RoboDK station: Project_AutomationPipeCouplingArm_Full.rdk

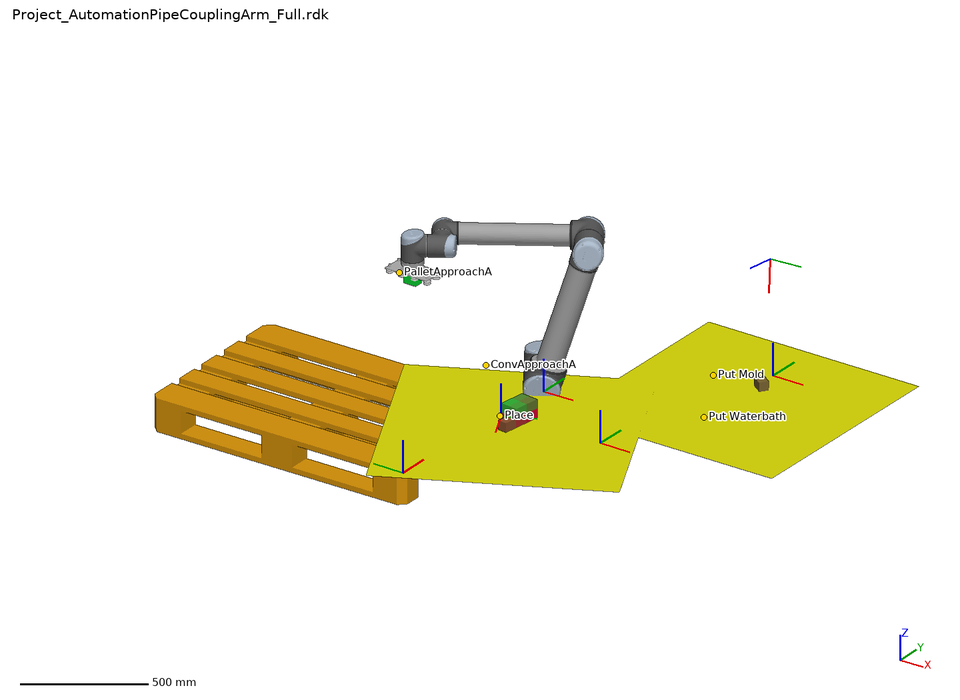
[picture v0: the station drawn from its stored meshes, robots at their saved joint values, targets as dots, program paths as lines]
Station Project_AutomationPipeCouplingArm_Full (saved by RoboDK 5.9.0). Poses are relative to the parent item; angles as X-Y-Z fixed-axis rotations.
Station parameters (name, value as stored): SizeBox, 40, 60, 40, SizePallet, 2,3,2, ConvSpeed, 15.0, SENSOR, 0
  - frame UR10 Base A at (0, -212.57, -10) mm
    - robot UR10 A: 6 axes, payload 10 kg, reach 1300 mm, repeatability 0.1 mm, weight 28.9 kg
        modified DH rows (alpha deg, a mm, theta deg, d mm): 0, 0, 0, 118; 90, 0, 180, 0; 0, 612.7, 0, 0; 0, 571.6, 0, 163.9; -90, 0, 0, 115.7; 90, 0, 180, 92.2
        joint limits [-360, -360, -360, -360, -360, -360] to [360, 360, 360, 360, 360, 360]; home [0, -90, 90, -90, -90, 0]; saved at [33.215, -107.184, 106.915, -89.731, -90, -55.617]
      - tool GripperA, TCP at (0, 0, 30) mm, rotated rx 0 ry 0 rz 90 deg, size 209.9 x 42 x 100 mm, geometry from test.iges
        - object Part 12 at (0, 0, 20) mm, rotated rx -180 ry 0 rz 0 deg, size 40 x 60 x 40 mm, geometry from box.sld
      - tool TCP A, TCP at (0, 0, 50) mm, rotated rx 0 ry 0 rz 90 deg
      - tool TCP A, TCP at (0, 0, 50) mm, rotated rx 0 ry 0 rz 90 deg
      - tool TCP A, TCP at (0, 0, 50) mm, rotated rx 0 ry 0 rz 90 deg
      - tool TCP A, TCP at (0, 0, 50) mm, rotated rx 0 ry 0 rz 90 deg
      - tool TCP A, TCP at (0, 0, 50) mm, rotated rx 0 ry 0 rz 90 deg
      - tool TCP A, TCP at (0, 0, 50) mm, rotated rx 0 ry 0 rz 90 deg
      - tool TCP A, TCP at (0, 0, 50) mm, rotated rx 0 ry 0 rz 90 deg
      - tool TCP A, TCP at (0, 0, 50) mm, rotated rx 0 ry 0 rz 90 deg
      - tool TCP A, TCP at (0, 0, 50) mm, rotated rx 0 ry 0 rz 90 deg
      - tool TCP A, TCP at (0, 0, 50) mm, rotated rx 0 ry 0 rz 90 deg
      - tool TCP A, TCP at (0, 0, 50) mm, rotated rx 0 ry 0 rz 90 deg
      - tool TCP A, TCP at (0, 0, 50) mm, rotated rx 0 ry 0 rz 90 deg
      - tool TCP A, TCP at (0, 0, 50) mm, rotated rx 0 ry 0 rz 90 deg
    - frame PalletA at (-344.62, -460.78, -266.49) mm, rotated rx 0 ry 0 rz 90.24 deg
      - object Europallet at (0, 0, 0) mm, size 800 x 144 x 1200 mm, geometry from User Library-Europallet.igs
      - object box100mm at (0, 0, 0) mm, size 100 x 100 x 100 mm, geometry from box.sld
    - target PalletApproachA (joint target) at (-397.36, -413.15, 569.38) mm, rotated rx 180 ry 0 rz 88.83 deg; joints [29.502, -102.797, 97.668, -84.871, -90, -59.329] of UR10 A
    - target ConvApproachA (joint target) at (568.44, -1202.75, 751.6) mm, rotated rx -180 ry -0.01 rz 172.23 deg; joints [75.247, -49.032, 15.798, -56.77, -90.009, -96.984] of UR10 A
  - frame WaterbathReference at (597.23, -679.82, 119.18) mm
    - target Put Waterbath (Cartesian target) at (200, 422.12, 0) mm, rotated rx -180 ry 0 rz 180 deg; joints [7.229, -35.446, 107.125, -161.679, -90, 96.985] of UR10 A
  - Python program SetSimulationParams (listed below)
  - Python program PrepareSimulation (listed below)
  - Python program SimulateCamera (listed below)
  - Python program PartsToWaterbath (listed below)
  - object Plane 1m x 1m at (787.21, 0, 87.75) mm, size 1000 x 1000 x 0.5 mm, geometry from plane.sld
  - camera Camera 1
  - camera Camera 2
  - frame Mold at (855.48, 127.88, 161.36) mm
    - object Part 6 at (-48.89, -11.25, -42.96) mm, rotated rx 0 ry -0.01 rz -124.63 deg, size 40 x 60 x 40 mm, geometry from box.sld
    - target Put Mold (Cartesian target) at (-210.52, -106.05, -13.69) mm, rotated rx -180 ry -0.01 rz 172.23 deg; joints [185.657, -70.282, 115.738, -135.446, -90, 13.426] of UR10 A
  - frame MoldApproach at (699.61, 332.1, 543.62) mm, rotated rx 7.77 ry 84.09 rz -81.21 deg
  - Python program PartsToMold (listed below)
  - object Plane 1m x 1m at (209.02, -727.11, 94.91) mm, rotated rx 0 ry 0 rz -63.61 deg, size 1000 x 1000 x 0.5 mm, geometry from plane.sld
  - frame Intermediate at (338.81, -986.14, 284.88) mm, rotated rx 0 ry 0 rz -63.14 deg
    - target Place (Cartesian target) at (-48.89, -11.25, -22.96) mm, rotated rx -180 ry -0.01 rz -124.63 deg; joints [100.774, -73.673, 104.377, -120.703, -90.01, -71.457] of UR10 A
    - object Part 10 at (-98.26, 22.85, -2.96) mm, rotated rx 0 ry -0.01 rz -124.63 deg, size 40 x 60 x 40 mm, geometry from box.sld
    - object Part 5 at (-26.16, 21.66, -42.96) mm, rotated rx 0 ry -0.01 rz -124.63 deg, size 40 x 60 x 40 mm, geometry from box.sld
    - object Part 9 at (-75.53, 55.76, -2.96) mm, rotated rx 0 ry -0.01 rz -124.63 deg, size 40 x 60 x 40 mm, geometry from box.sld
    - object Part 3 at (-75.53, 55.76, -42.96) mm, rotated rx 0 ry -0.01 rz -124.63 deg, size 40 x 60 x 40 mm, geometry from box.sld
    - object Part 4 at (-98.26, 22.84, -42.96) mm, rotated rx 0 ry -0.01 rz -124.63 deg, size 40 x 60 x 40 mm, geometry from box.sld
    - camera Camera 3
    - object Part 7 at (-124.9, 89.86, -2.97) mm, rotated rx 0 ry -0.01 rz -124.63 deg, size 40 x 60 x 40 mm, geometry from box.sld
    - object Part 8 at (-147.63, 56.94, -2.96) mm, rotated rx 0 ry -0.01 rz -124.63 deg, size 40 x 60 x 40 mm, geometry from box.sld
    - object Part 2 at (-147.64, 56.94, -42.96) mm, rotated rx 0 ry -0.01 rz -124.63 deg, size 40 x 60 x 40 mm, geometry from box.sld
    - object Part 1 at (-124.91, 89.85, -42.97) mm, rotated rx 0 ry -0.01 rz -124.63 deg, size 40 x 60 x 40 mm, geometry from box.sld
  - Python program Prog6 (listed below)
  - Python program Prog7 (listed below)
  - Python program Prog8 (listed below)

--- Python program SetSimulationParams ---
# Type help("robolink") or help("robodk") for more information
# Press F5 to run the script
# Note: you do not need to keep a copy of this file, your python script is saved with the station
from robolink import *    # API to communicate with RoboDK
from robodk import *      # basic matrix operations


PARAM_SIZE_BOX = 'SizeBox'
PARAM_SIZE_PALLET = 'SizePallet'
PARAM_CONV_SPEED_MM = 'ConvSpeed'



RDK = Robolink()

size_box = RDK.getParam(PARAM_SIZE_BOX)
size_pallet = RDK.getParam(PARAM_SIZE_PALLET)
conv_speed = RDK.getParam(PARAM_CONV_SPEED_MM)

# ------------------------------------------------------------
size_box_input = mbox('Enter the size of the box in mm [L,W,H]', entry=size_box)
if size_box_input:
    RDK.setParam(PARAM_SIZE_BOX, size_box_input)
else:
    raise Exception('Operation cancelled by user')

# ------------------------------------------------------------
size_pallet_input = mbox('Enter the size of the pallet', entry=size_pallet)
if size_pallet_input:
    RDK.setParam(PARAM_SIZE_PALLET, size_pallet_input)
else:
    raise Exception('Operation cancelled by user')

# ------------------------------------------------------------
conv_speed_input = mbox('Enter the speed of the conveyor in mm/s', entry=conv_speed)
if conv_speed_input:
    RDK.setParam(PARAM_CONV_SPEED_MM, conv_speed_input)
    conv_speed = float(conv_speed_input)
    conv = RDK.Item('Conveyor Belt', ITEM_TYPE_ROBOT)
    conv.setSpeed(conv_speed)

else:
    raise Exception('Operation cancelled by user')

--- Python program PrepareSimulation ---
# Type help("robolink") or help("robodk") for more information
# Press F5 to run the script
# Note: you do not need to keep a copy of this file, your python script is saved with the station
from robolink import *    # API to communicate with RoboDK
from robodk import *      # basic matrix operations

# Use RoboDK API as RL
RDK = Robolink()

frame_pallet        = RDK.Item('PalletA', ITEM_TYPE_FRAME)

# get variable parameters
SIZE_BOX = RDK.getParam('SizeBox')
SIZE_PALLET = RDK.getParam('SizePallet')
SIZE_BOX_XYZ = [float(x.replace(' ','')) for x in SIZE_BOX.split(',')]
SIZE_PALLET_XYZ = [float(x.replace(' ','')) for x in SIZE_PALLET.split(',')]
SIZE_BOX_Z = SIZE_BOX_XYZ[2] # the height of the boxes is important to take into account when approaching the positions

def box_calc(size_xyz, pallet_xyz):
    """Calculates a list of points to store parts in a pallet"""
    [size_x, size_y, size_z] = size_xyz
    [pallet_x, pallet_y, pallet_z] = pallet_xyz
    xyz_list = []
    for h in range(int(pallet_z)):
        for j in range(int(pallet_y)):
            for i in range(int(pallet_x)):
                xyz_list = xyz_list + [[(i+0.5)*size_x, (j+0.5)*size_y, (h+0.5)*size_z]]
    return xyz_list

def parts_setup(frame, positions, size_xyz):
    """Place a list of parts in a reference frame. The part/reference object must have been previously copied to the clipboard."""
    [size_x, size_y, size_z] = size_xyz
    nparts = len(positions)
    cstep = 1.0/(nparts - 1)
    for i in range(nparts):
        newpart = frame.Paste()
        newpart.Scale([size_x/100, size_y/100, size_z/100]) #scale with respect to the reference object (100mm cube)
        newpart.setName('Part ' + str(i+1)) #set item name
        newpart.setPose(transl(positions[i])) #set item position with respect to parent
        newpart.setVisible(True, False) #make item visible but hide the reference frame
        newpart.Recolor([1-cstep*i, cstep*i, 0.2, 1]) #set RGBA color

def cleanup(objects, startswith="Part "):
    """Deletes all objects where the name starts with "startswith", from the provided list of objects."""
    for item in objects:
        if item.Name().startswith(startswith):
            item.Delete()

# turn off rendering (much faster when setting up the station)
RDK.Render(False)

# cleanup previous simulation (generated parts and tools)
all_objects = RDK.ItemList(ITEM_TYPE_OBJECT, False)
cleanup(all_objects, 'Part ')
all_tools = RDK.ItemList(ITEM_TYPE_TOOL, False)
cleanup(all_tools, 'TCP ')

# copy the reference part
partref = RDK.Item('box100mm')
partref.Copy()

#RL.Set_Simulation_Speed(500);
#RL.Set_Simulation_Mode(1)

# calculate an array of positions to get/store the parts
parts_positions = box_calc(SIZE_BOX_XYZ, SIZE_PALLET_XYZ)

# setup/initialise the parts on the palled
parts_setup(frame_pallet, parts_positions, SIZE_BOX_XYZ)

RDK.Render(True)

--- Python program SimulateCamera ---
# Type help("robolink") or help("robodk") for more information
# Press F5 to run the script
# Note: you do not need to keep a copy of this file, your python script is saved with the station
from robolink import *    # API to communicate with RoboDK
from robodk import *      # basic matrix operations
RDK = Robolink()

# Close any open 2D camera views
RDK.Cam2D_Close()

camref = RDK.Item('Camera Reference',ITEM_TYPE_FRAME)

# set parameters in mm and degrees:
# FOV: Field of view in degrees (atan(0.5*height/distance) of the sensor divided by
# FOCAL_LENGHT: focal lenght in mm
# FAR_LENGHT: maximum working distance (in mm)
# SIZE: size of the sensor in pixels
# BG_COLOR: background color (rgb color or named color: AARRGGBB)
# LIGHT_AMBIENT: ambient color (rgb color or named color: AARRGGBB)
# LIGHT_SPECULAR: specular color (rgb color or named color: AARRGGBB)
# LIGHT_DIFFUSE: diffuse color (rgb color or named color: AARRGGBB)


# cam_id = RDK.Cam2D_Add(camref, 'FOCAL_LENGHT=6 FOV=32 FAR_LENGHT=1000 SIZE=640x480 BG_COLOR=black')
# cam_id = RDK.Cam2D_Add(camref, 'FOCAL_LENGHT=6 FOV=32 FAR_LENGHT=1000 SIZE=640x480')
# cam_id = RDK.Cam2D_Add(camref, 'FOCAL_LENGHT=6 FOV=32 FAR_LENGHT=1000 SIZE=640x480 BG_COLOR=black LIGHT_AMBIENT=red LIGHT_DIFFUSE=#FF00FF00 LIGHT_SPECULAR=black')
# cam_id = RDK.Cam2D_Add(camref, 'FOCAL_LENGHT=6 FOV=32 FAR_LENGHT=1000 SIZE=640x480 DEPTH')
cam_id = RDK.Cam2D_Add(camref, 'FOCAL_LENGHT=6 FOV=32 FAR_LENGHT=1000 SIZE=640x480 BG_COLOR=black LIGHT_AMBIENT=red LIGHT_DIFFUSE=black LIGHT_SPECULAR=white')


# cam_id = RDK.Cam2D_Add(camref, 'FOCAL_LENGHT=6 FOV=32 FAR_LENGHT=1000 SIZE=640x480 LIGHT_AMBIENT=red')

# cam_id = RDK.Cam2D_Add(camref, 'POPUP')

# RDK.Cam2D_Snapshot(RDK.getParam('PATH_OPENSTATION') + "/sample_image.png", cam_id)

--- Python program PartsToWaterbath ---
# Type help("robolink") or help("robodk") for more information
# Press F5 to run the script
# Note: you do not need to keep a copy of this file, your python script is saved with the station
from robolink import *    # API to communicate with RoboDK
from robodk import *      # basic matrix operations
from random import uniform

# Use RoboDK API as RL
RDK = Robolink()

# define default approach distance
APPROACH = 100

# gather robot, tool and reference frames from the station
robot               = RDK.Item('UR10 A', ITEM_TYPE_ROBOT)
tool                = RDK.Item('GripperA', ITEM_TYPE_TOOL)
frame_pallet        = RDK.Item('PalletA', ITEM_TYPE_FRAME)
frame_conv          = RDK.Item('ConveyorReference', ITEM_TYPE_FRAME)
frame_conv_moving   = RDK.Item('MovingRef', ITEM_TYPE_FRAME)

# gather targets
target_pallet_safe = RDK.Item('PalletApproachA', ITEM_TYPE_TARGET)
target_conv_safe = RDK.Item('ConvApproachA', ITEM_TYPE_TARGET)
target_conv = RDK.Item('Put Conveyor', ITEM_TYPE_TARGET)

# get variable parameters
SIZE_BOX = RDK.getParam('SizeBox')
SIZE_PALLET = RDK.getParam('SizePallet')
SIZE_BOX_XYZ = [float(x.replace(' ','')) for x in SIZE_BOX.split(',')]
SIZE_PALLET_XYZ = [float(x.replace(' ','')) for x in SIZE_PALLET.split(',')]
SIZE_BOX_Z = SIZE_BOX_XYZ[2] # the height of the boxes is important to take into account when approaching the positions

def box_calc(size_xyz, pallet_xyz):
    """Calculates a list of points to store parts in a pallet"""
    [size_x, size_y, size_z] = size_xyz
    [pallet_x, pallet_y, pallet_z] = pallet_xyz
    xyz_list = []
    for h in range(int(pallet_z)):
        for j in range(int(pallet_y)):
            for i in range(int(pallet_x)):
                xyz_list = xyz_list + [[(i+0.5)*size_x, (j+0.5)*size_y, (h+0.5)*size_z]]
    return xyz_list

def TCP_On(toolitem):
    """Attaches the closest object to the toolitem Htool pose,
    It will also output appropriate function calls on the generated robot program (call to TCP_On)"""
    toolitem.AttachClosest()
    toolitem.RDK().RunMessage('Set air valve on')
    toolitem.RDK().RunProgram('TCP_On()');

def TCP_Off(toolitem, itemleave=0):
    """Detaches the closest object attached to the toolitem Htool pose,
    It will also output appropriate function calls on the generated robot program (call to TCP_Off)"""
    toolitem.DetachAll(itemleave)
    toolitem.RDK().RunMessage('Set air valve off')
    toolitem.RDK().RunProgram('TCP_Off()');

#RL.Set_Simulation_Speed(500);
#RL.Set_Simulation_Mode(1)

# calculate an array of positions to get/store the parts
parts_positions = box_calc(SIZE_BOX_XYZ, SIZE_PALLET_XYZ)

# Calculate a new TCP that takes into account the size of the part (targets are set to the center of the box)
tool_xyzrpw = tool.PoseTool()*transl(0,0,SIZE_BOX_Z/2)
tool_tcp = robot.AddTool(tool_xyzrpw, 'TCP A')

# ---------------------------------------------------------------------------------
# -------------------------- PROGRAM START ----------------------------------------

robot.setPoseTool(tool_tcp)
nparts = len(parts_positions)
i = nparts-1
while i >= 0:
    # ----------- take a part from the pallet ------
    # get the xyz position of part i
    robot.setPoseFrame(frame_pallet)
    part_position_i = parts_positions[i]
    target_i = transl(part_position_i)*rotx(pi)
    target_i_app = target_i * transl(0,0,-(APPROACH+SIZE_BOX_Z))
    # approach to the pallet
    robot.MoveJ(target_pallet_safe)
    # get the box i
    robot.MoveJ(target_i_app)
    robot.MoveL(target_i)
    TCP_On(tool) # attach the closest part
    robot.MoveL(target_i_app)
    robot.MoveJ(target_pallet_safe)

    # ----------- place the box i on the convegor ------
    # approach to the conveyor
    robot.setPoseFrame(frame_conv)
    target_conv_pose = target_conv.Pose()*transl(0,0,-SIZE_BOX_Z/2)
    target_conv_app = target_conv_pose*transl(0,0,-APPROACH)
    robot.MoveJ(target_conv_safe)
    robot.MoveJ(target_conv_app)

    # Place the part at a random position with respect to the target on the conveyor
    TX = uniform(-150, 150)
    RZ = uniform(-90*pi/180, +90*pi/180)

    robot.MoveL(target_conv_pose*transl(TX,0,0)*rotz(RZ))
    TCP_Off(tool, frame_conv_moving) # detach an place the object in the moving reference frame of the conveyor
    robot.MoveL(target_conv_app)
    robot.MoveJ(target_conv_safe)

    i = i - 1

--- Python program PartsToMold ---
# PartsToMold.py
from robolink import *    # API to communicate with RoboDK
from robodk import *      # basic matrix operations
from random import uniform

# Connect to RoboDK
RDK = Robolink()

# Define constants
APPROACH = 100

# Retrieve robot, tool, and frames
robot               = RDK.Item('UR10 A', ITEM_TYPE_ROBOT)
tool                = RDK.Item('GripperA', ITEM_TYPE_TOOL)
frame_conv_moving   = RDK.Item('MovingRef', ITEM_TYPE_FRAME)
frame_mold          = RDK.Item('Mold', ITEM_TYPE_FRAME)

# Retrieve targets
target_conv_safe = RDK.Item('ConvApproachA', ITEM_TYPE_TARGET)
target_conv       = RDK.Item('Put Conveyor', ITEM_TYPE_TARGET)
target_mold_safe  = RDK.Item('MoldApproach', ITEM_TYPE_TARGET)
target_mold       = RDK.Item('Put Mold', ITEM_TYPE_TARGET)

# Get box size parameter
SIZE_BOX = RDK.getParam('SizeBox')
SIZE_BOX_XYZ = [float(x.replace(' ','')) for x in SIZE_BOX.split(',')]
SIZE_BOX_Z = SIZE_BOX_XYZ[2]  # Height of the box

# Define TCP that includes half the box height
tool_xyzrpw = tool.PoseTool()*transl(0,0,SIZE_BOX_Z/2)
tool_tcp = robot.AddTool(tool_xyzrpw, 'TCP A')
robot.setPoseTool(tool_tcp)

def TCP_On(toolitem):
    """Attach part to tool."""
    toolitem.AttachClosest()
    toolitem.RDK().RunMessage('Set air valve on')
    toolitem.RDK().RunProgram('TCP_On()')

def TCP_Off(toolitem, itemleave=0):
    """Detach part from tool."""
    toolitem.DetachAll(itemleave)
    toolitem.RDK().RunMessage('Set air valve off')
    toolitem.RDK().RunProgram('TCP_Off()')

# ----------------------------- PROGRAM START -----------------------------

# You can loop over multiple parts if needed; here we do it once
robot.setPoseFrame(frame_conv_moving)

# Approach conveyor
target_conv_pose = target_conv.Pose()*transl(0,0,-SIZE_BOX_Z/2)
target_conv_app = target_conv_pose*transl(0,0,-APPROACH)

robot.MoveJ(target_conv_safe)
robot.MoveJ(target_conv_app)

# Simulate random pick offset (in case conveyor is moving)
TX = uniform(-150, 150)
RZ = uniform(-90*pi/180, +90*pi/180)
pickup_pose = target_conv_pose*transl(TX,0,0)*rotz(RZ)

robot.MoveL(pickup_pose)
TCP_On(tool)
robot.MoveL(target_conv_app)
robot.MoveJ(target_conv_safe)

# Move to mold
robot.setPoseFrame(frame_mold)

target_mold_pose = target_mold.Pose()*transl(0,0,-SIZE_BOX_Z/2)
target_mold_app = target_mold_pose*transl(0,0,-APPROACH)

robot.MoveJ(target_mold_safe)
robot.MoveJ(target_mold_app)
robot.MoveL(target_mold_pose)
TCP_Off(tool, frame_mold)
robot.MoveL(target_mold_app)
robot.MoveJ(target_mold_safe)

--- Python program Prog6 ---
from robolink import *    # API to communicate with RoboDK
from robodk import *      # basic matrix operations
from random import uniform

# Initialize RoboDK API
RDK = Robolink()

# Default approach distance
APPROACH = 100

# Gather robot, tool and frames
robot               = RDK.Item('UR10 A', ITEM_TYPE_ROBOT)
tool                = RDK.Item('GripperA', ITEM_TYPE_TOOL)
frame_pallet        = RDK.Item('PalletA', ITEM_TYPE_FRAME)
frame_conv          = RDK.Item('ConveyorReference', ITEM_TYPE_FRAME)
frame_conv_moving   = RDK.Item('MovingRef', ITEM_TYPE_FRAME)
frame_intermediate  = RDK.Item('Intermediate', ITEM_TYPE_FRAME)

# Gather targets
target_pallet_safe  = RDK.Item('PalletApproachA', ITEM_TYPE_TARGET)
target_conv_safe    = RDK.Item('ConvApproachA', ITEM_TYPE_TARGET)
target_conv         = RDK.Item('Put Conveyor', ITEM_TYPE_TARGET)
target_place        = RDK.Item('Place', ITEM_TYPE_TARGET)

# Get box and pallet dimensions
SIZE_BOX = RDK.getParam('SizeBox')
SIZE_PALLET = RDK.getParam('SizePallet')
SIZE_BOX_XYZ = [float(x.replace(' ','')) for x in SIZE_BOX.split(',')]
SIZE_PALLET_XYZ = [float(x.replace(' ','')) for x in SIZE_PALLET.split(',')]
SIZE_BOX_Z = SIZE_BOX_XYZ[2]

# Function to calculate pallet positions
def box_calc(size_xyz, pallet_xyz):
    [size_x, size_y, size_z] = size_xyz
    [pallet_x, pallet_y, pallet_z] = pallet_xyz
    xyz_list = []
    for h in range(int(pallet_z)):
        for j in range(int(pallet_y)):
            for i in range(int(pallet_x)):
                xyz_list.append([(i+0.5)*size_x, (j+0.5)*size_y, (h+0.5)*size_z])
    return xyz_list

# Attach part to tool
def TCP_On(toolitem):
    toolitem.AttachClosest()
    toolitem.RDK().RunMessage('Set air valve on')
    toolitem.RDK().RunProgram('TCP_On()');

# Detach part from tool
def TCP_Off(toolitem, itemleave=0):
    toolitem.DetachAll(itemleave)
    toolitem.RDK().RunMessage('Set air valve off')
    toolitem.RDK().RunProgram('TCP_Off()');

# Calculate part positions
parts_positions = box_calc(SIZE_BOX_XYZ, SIZE_PALLET_XYZ)

# Create adjusted TCP for grasping center
tool_xyzrpw = tool.PoseTool() * transl(0, 0, SIZE_BOX_Z/2)
tool_tcp = robot.AddTool(tool_xyzrpw, 'TCP A')

# Start main program
robot.setPoseTool(tool_tcp)
nparts = len(parts_positions)
i = nparts - 1

while i >= 0:
    # ----------- Take part from pallet -----------
    robot.setPoseFrame(frame_pallet)
    part_position_i = parts_positions[i]
    target_i = transl(part_position_i) * rotx(pi)
    target_i_app = target_i * transl(0, 0, -(APPROACH + SIZE_BOX_Z))

    robot.MoveJ(target_pallet_safe)
    robot.MoveJ(target_i_app)
    robot.MoveL(target_i)
    TCP_On(tool)
    robot.MoveL(target_i_app)
    robot.MoveJ(target_pallet_safe)

    # ----------- Temporarily place in Intermediate frame -----------
    robot.setPoseFrame(frame_intermediate)
    target_place_pose = target_place.Pose() * transl(0, 0, -SIZE_BOX_Z/2)
    target_place_app = target_place_pose * transl(0, 0, -APPROACH)

    robot.MoveJ(target_place_app)
    robot.MoveL(target_place_pose)
    TCP_Off(tool, frame_intermediate)
    robot.MoveL(target_place_app)

    pause(2)  # Wait for 2 seconds

    # ----------- Pick back from Intermediate frame -----------
    robot.MoveJ(target_place_app)
    robot.MoveL(target_place_pose)
    TCP_On(tool)
    robot.MoveL(target_place_app)

    # ----------- Final placement on conveyor -----------
    robot.setPoseFrame(frame_conv)
    target_conv_pose = target_conv.Pose() * transl(0, 0, -SIZE_BOX_Z/2)
    target_conv_app = target_conv_pose * transl(0, 0, -APPROACH)

    robot.MoveJ(target_conv_safe)
    robot.MoveJ(target_conv_app)

    TX = uniform(-150, 150)
    RZ = uniform(-90*pi/180, +90*pi/180)

    robot.MoveL(target_conv_pose * transl(TX, 0, 0) * rotz(RZ))
    TCP_Off(tool, frame_conv_moving)
    robot.MoveL(target_conv_app)
    robot.MoveJ(target_conv_safe)

    i = i - 1

--- Python program Prog7 ---
from robolink import *    # API to communicate with RoboDK
from robodk import *      # basic matrix operations
from random import uniform
import time

# Connect to RoboDK
RDK = Robolink()

APPROACH = 100

# Items from the station
robot               = RDK.Item('UR10 A', ITEM_TYPE_ROBOT)
tool                = RDK.Item('GripperA', ITEM_TYPE_TOOL)
frame_pallet        = RDK.Item('PalletA', ITEM_TYPE_FRAME)
frame_intermediate  = RDK.Item('Intermediate', ITEM_TYPE_FRAME)
frame_final         = RDK.Item('Mold', ITEM_TYPE_FRAME)

# Targets
target_pallet_safe = RDK.Item('PalletApproachA', ITEM_TYPE_TARGET)
target_place       = RDK.Item('Place', ITEM_TYPE_TARGET)
target_final       = RDK.Item('Put Mold', ITEM_TYPE_TARGET)
target_final_safe  = RDK.Item('MoldApproach', ITEM_TYPE_TARGET)

# Parameter values
SIZE_BOX = RDK.getParam('SizeBox')
SIZE_PALLET = RDK.getParam('SizePallet')
SIZE_BOX_XYZ = [float(x.strip()) for x in SIZE_BOX.split(',')]
SIZE_PALLET_XYZ = [float(x.strip()) for x in SIZE_PALLET.split(',')]
SIZE_BOX_Z = SIZE_BOX_XYZ[2]

# Tool TCP considering box height
tool_xyzrpw = tool.PoseTool() * transl(0, 0, SIZE_BOX_Z / 2)
tool_tcp = robot.AddTool(tool_xyzrpw, 'TCP A')
robot.setPoseTool(tool_tcp)

# Function to compute pallet box positions
def box_calc(size_xyz, pallet_xyz):
    [size_x, size_y, size_z] = size_xyz
    [pallet_x, pallet_y, pallet_z] = pallet_xyz
    xyz_list = []
    for h in range(int(pallet_z)):
        for j in range(int(pallet_y)):
            for i in range(int(pallet_x)):
                xyz_list += [[(i+0.5)*size_x, (j+0.5)*size_y, (h+0.5)*size_z]]
    return xyz_list

# Gripper control
def TCP_On(toolitem):
    toolitem.AttachClosest()
    RDK.RunMessage('Set air valve on')
    RDK.RunProgram('TCP_On()')

def TCP_Off(toolitem, itemleave=0):
    toolitem.DetachAll(itemleave)
    RDK.RunMessage('Set air valve off')
    RDK.RunProgram('TCP_Off()')

# Get box positions
parts_positions = box_calc(SIZE_BOX_XYZ, SIZE_PALLET_XYZ)

# Start program
nparts = len(parts_positions)
i = nparts - 1

while i >= 0:
    # -------- PICK from Pallet --------
    robot.setPoseFrame(frame_pallet)
    part_position_i = parts_positions[i]
    target_i = transl(part_position_i) * rotx(pi)
    target_i_app = target_i * transl(0, 0, -(APPROACH + SIZE_BOX_Z))

    robot.MoveJ(target_pallet_safe)
    robot.MoveJ(target_i_app)
    robot.MoveL(target_i)
    TCP_On(tool)
    robot.MoveL(target_i_app)
    robot.MoveJ(target_pallet_safe)

    # -------- PLACE at Intermediate --------
    robot.setPoseFrame(frame_intermediate)
    target_place_pose = target_place.Pose() * transl(0, 0, -SIZE_BOX_Z / 2)
    target_place_app = target_place_pose * transl(0, 0, -APPROACH)

    robot.MoveJ(target_place_app)
    robot.MoveL(target_place_pose)
    TCP_Off(tool, frame_intermediate)  # leave object
    robot.MoveL(target_place_app)
    robot.MoveJ(target_pallet_safe)

    time.sleep(2)  # Wait for 2 seconds

    # -------- PICK BACK from Intermediate --------
    robot.MoveJ(target_place_app)
    robot.MoveL(target_place_pose)
    TCP_On(tool)  # Pick object again
    robot.MoveL(target_place_app)
    robot.MoveJ(target_pallet_safe)

    # -------- PLACE at Final Destination (Mold) --------
    robot.setPoseFrame(frame_final)
    target_final_pose = target_final.Pose() * transl(0, 0, -SIZE_BOX_Z / 2)
    target_final_app = target_final_pose * transl(0, 0, -APPROACH)

    robot.MoveJ(target_final_safe)
    robot.MoveJ(target_final_app)
    robot.MoveL(target_final_pose)
    TCP_Off(tool, frame_final)
    robot.MoveL(target_final_app)
    robot.MoveJ(target_final_safe)

    i -= 1

--- Python program Prog8 ---
from robolink import *    # API to communicate with RoboDK
from robodk import *      # basic matrix operations
from random import uniform
import time

# Connect to RoboDK
RDK = Robolink()

APPROACH = 100

# Items from the station
robot               = RDK.Item('UR10 A', ITEM_TYPE_ROBOT)
tool                = RDK.Item('GripperA', ITEM_TYPE_TOOL)
frame_pallet        = RDK.Item('PalletA', ITEM_TYPE_FRAME)
frame_intermediate  = RDK.Item('Intermediate', ITEM_TYPE_FRAME)
frame_final         = RDK.Item('Mold', ITEM_TYPE_FRAME)

# Targets
target_pallet_safe = RDK.Item('PalletApproachA', ITEM_TYPE_TARGET)
target_place       = RDK.Item('Place', ITEM_TYPE_TARGET)
target_final       = RDK.Item('Put Mold', ITEM_TYPE_TARGET)
target_final_safe  = RDK.Item('MoldApproach', ITEM_TYPE_TARGET)

# Parameter values
SIZE_BOX = RDK.getParam('SizeBox')
SIZE_PALLET = RDK.getParam('SizePallet')
SIZE_BOX_XYZ = [float(x.strip()) for x in SIZE_BOX.split(',')]
SIZE_PALLET_XYZ = [float(x.strip()) for x in SIZE_PALLET.split(',')]
SIZE_BOX_Z = SIZE_BOX_XYZ[2]

# Tool TCP considering box height
tool_xyzrpw = tool.PoseTool() * transl(0, 0, SIZE_BOX_Z / 2)
tool_tcp = robot.AddTool(tool_xyzrpw, 'TCP A')
robot.setPoseTool(tool_tcp)

# Function to compute pallet box positions
def box_calc(size_xyz, pallet_xyz):
    [size_x, size_y, size_z] = size_xyz
    [pallet_x, pallet_y, pallet_z] = pallet_xyz
    xyz_list = []
    for h in range(int(pallet_z)):
        for j in range(int(pallet_y)):
            for i in range(int(pallet_x)):
                xyz_list += [[(i+0.5)*size_x, (j+0.5)*size_y, (h+0.5)*size_z]]
    return xyz_list

# Gripper control
def TCP_On(toolitem):
    toolitem.AttachClosest()
    RDK.RunMessage('Set air valve on')
    RDK.RunProgram('TCP_On()')

def TCP_Off(toolitem, itemleave=0):
    toolitem.DetachAll(itemleave)
    RDK.RunMessage('Set air valve off')
    RDK.RunProgram('TCP_Off()')

# Get box positions
parts_positions = box_calc(SIZE_BOX_XYZ, SIZE_PALLET_XYZ)

# Start program
nparts = len(parts_positions)
i = nparts - 1

while i >= 0:
    # -------- PICK from Pallet --------
    robot.setPoseFrame(frame_pallet)
    part_position_i = parts_positions[i]
    target_i = transl(part_position_i) * rotx(pi)
    target_i_app = target_i * transl(0, 0, -(APPROACH + SIZE_BOX_Z))

    robot.MoveJ(target_pallet_safe)
    robot.MoveJ(target_i_app)
    robot.MoveL(target_i)
    TCP_On(tool)
    robot.MoveL(target_i_app)
    robot.MoveJ(target_pallet_safe)

    # -------- PLACE at Intermediate --------
    robot.setPoseFrame(frame_intermediate)
    target_place_pose = target_place.Pose() * transl(0, 0, -SIZE_BOX_Z / 2)
    target_place_app = target_place_pose * transl(0, 0, -APPROACH)

    robot.MoveJ(target_place_app)
    robot.MoveL(target_place_pose)
    TCP_Off(tool, frame_intermediate)  # Leave object at intermediate
    robot.MoveL(target_place_app)
    robot.MoveJ(target_pallet_safe)

    # -------- WAIT for 2 seconds --------
    time.sleep(2)

    # -------- PICK BACK from Intermediate --------
    robot.setPoseFrame(frame_intermediate)
    robot.MoveJ(target_place_app)
    robot.MoveL(target_place_pose)
    TCP_On(tool)  # Pick object again
    robot.MoveL(target_place_app)
    robot.MoveJ(target_pallet_safe)

    # -------- PLACE at Final Destination (Mold) --------
    robot.setPoseFrame(frame_final)
    target_final_pose = target_final.Pose() * transl(0, 0, -SIZE_BOX_Z / 2)
    target_final_app = target_final_pose * transl(0, 0, -APPROACH)

    robot.MoveJ(target_final_safe)
    robot.MoveJ(target_final_app)
    robot.MoveL(target_final_pose)
    TCP_Off(tool, frame_final)  # Leave object at final
    robot.MoveL(target_final_app)
    robot.MoveJ(target_final_safe)

    i -= 1
